INTERFACE I_Process_LinkedList

METHOD AddHeadValue : ST_PROCESS_LIST_RESULT
VAR_INPUT
  stData        : ST_PROCESS_DATA;
END_VAR
END_METHOD

METHOD AddTailValue : ST_PROCESS_LIST_RESULT
VAR_INPUT
  stData        : ST_PROCESS_DATA;
END_VAR
END_METHOD

PROPERTY Count : UDINT
GET
END_GET
END_PROPERTY

PROPERTY Data : ARRAY[1..MAX_LIST_NODES] OF ST_PROCESS_DATA
GET
END_GET
END_PROPERTY

PROPERTY Free : UDINT
GET
END_GET
END_PROPERTY

METHOD GetHead : ST_PROCESS_LIST_RESULT
VAR_INPUT
END_VAR
END_METHOD

METHOD GetTail : ST_PROCESS_LIST_RESULT
VAR_INPUT
END_VAR
VAR
END_VAR
END_METHOD

METHOD InitList : BOOL
END_METHOD

PROPERTY Nodes : ARRAY[0..MAX_LIST_NODES] OF T_LinkedListEntry
GET
END_GET
END_PROPERTY

METHOD RemoveHeadValue : ST_PROCESS_LIST_RESULT
VAR_INPUT
END_VAR
END_METHOD

METHOD RemoveTailValue : ST_PROCESS_LIST_RESULT
VAR_INPUT
END_VAR
VAR
END_VAR
END_METHOD

END_INTERFACE

(* stored: Version 1.1.0.1
   Itf I_Process_LinkedList: Id {c6506b67-74dd-453a-a5aa-e797256a65a6}
   Method AddHeadValue: Id {8450ad0c-27f4-4ade-8398-39ad970d46c5}
   Method AddTailValue: Id {facfa38e-e691-458f-8658-f59a31b38cd2}
   Property Count: Id {4ae5812d-2455-4957-b637-cb08efe9d9fa}
   Get Get: Id {b84251db-7daa-44b8-945b-5ad8d1a3941e}
   Property Data: Id {9c656936-6238-44f2-b712-3b2c0205875c}
   Get Get: Id {c3ebf75f-8b52-42ae-983b-37bcb5a26609}
   Property Free: Id {2378d969-c423-4413-ba7b-b23047349907}
   Get Get: Id {5106e45b-d120-454e-a898-5044c80f0ed5}
   Method GetHead: Id {7162edae-85f9-4f2b-bcd7-0e99527e6211}
   Method GetTail: Id {ebd827ea-d9d2-4d8f-b428-fb54c8341f42}
   Method InitList: Id {ddbf3f45-9fb4-472c-bdbc-1b0931e07c2a}
   Property Nodes: Id {9c574555-200a-4497-b3f9-eb257067a9ea}
   Get Get: Id {3301d776-e4ef-4966-a5e3-e411f44da643}
   Method RemoveHeadValue: Id {179dbd5d-0cec-4c36-9ed8-91564477a269}
   Method RemoveTailValue: Id {0d030a16-c812-4d66-8d70-c63c29715f6a} *)
